FUNCTION_BLOCK CmdCAerationValves (* CAT Function Block Type *)
  (* Standard: 61499-2 *)
  (* Version 0.0, 6/8/2026, Schneider Electric, template *)
  PACKAGE SE.Nereda;
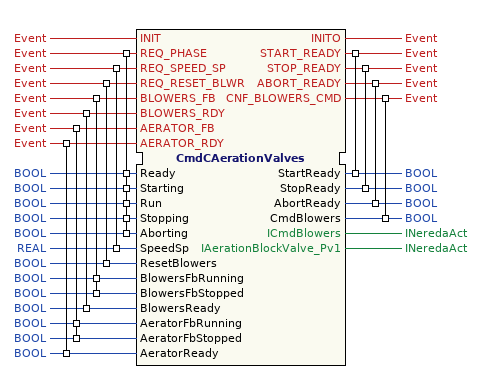
  EVENT_INPUT
    INIT;
    REQ_PHASE WITH Ready, Starting, Run, Stopping, Aborting;
    REQ_SPEED_SP WITH SpeedSp;
    REQ_RESET_BLWR WITH ResetBlowers;
    BLOWERS_FB WITH BlowersFbRunning, BlowersFbStopped;
    BLOWERS_RDY WITH BlowersReady;
    AERATOR_FB WITH AeratorFbRunning, AeratorFbStopped;
    AERATOR_RDY WITH AeratorReady;
  END_EVENT
  EVENT_OUTPUT
    INITO;
    START_READY WITH StartReady;
    STOP_READY WITH StopReady;
    ABORT_READY WITH AbortReady;
    CNF_BLOWERS_CMD WITH CmdBlowers;
  END_EVENT
  VAR_INPUT
    Ready : BOOL;
    Starting : BOOL;
    Run : BOOL;
    Stopping : BOOL;
    Aborting : BOOL;
    SpeedSp : REAL;
    ResetBlowers : BOOL;
    BlowersFbRunning : BOOL;
    BlowersFbStopped : BOOL;
    BlowersReady : BOOL;
    AeratorFbRunning : BOOL;
    AeratorFbStopped : BOOL;
    AeratorReady : BOOL;
  END_VAR
  VAR_OUTPUT
    StartReady : BOOL;
    StopReady : BOOL;
    AbortReady : BOOL;
    CmdBlowers : BOOL;
  END_VAR
  PLUGS
    ICmdBlowers : INeredaAct;
    IAerationBlockValve_Pv1 : INeredaAct;
  END_PLUGS
  (* 01 - FUNCTIONNAL INPUT INTERFACE *)
  (* 00 - INITIALIZATION *)
  (* 05 - LOGIC *)
  (* 06 - HMI INTERFACE *)
  (* 03 - FIELD INTERFACE *)
  (* 02 - FUNCTIONNAL OUTPUT INTERFACE *)
  (* Command Logic *)
  FBS
    IThis : CmdCAerationValves_HMI(QI := TRUE);
    CmdBlowersSmooth : boolValueChanged;
    FbRunBlowers : DS_SELECTX_2536758B411A6CE51; {SET_ATTRIBUTE(Configuration.GenericFBType.InterfaceParams, Runtime.Standard#CNTX:=2;CNTY:=1;DI${CNTX,_,CNTY$}:BOOL)}
    FbStopBlowers : DS_SELECTX_2536758B411A6CE51; {SET_ATTRIBUTE(Configuration.GenericFBType.InterfaceParams, Runtime.Standard#CNTX:=2;CNTY:=1;DI${CNTX,_,CNTY$}:BOOL)}
    FbReadyBlowers : DS_SELECTX_2536758B411A6CE51; {SET_ATTRIBUTE(Configuration.GenericFBType.InterfaceParams, Runtime.Standard#CNTX:=2;CNTY:=1;DI${CNTX,_,CNTY$}:BOOL)}
    BlowersCmd : BOOL2INT;
    CmdLogic : CmdCAerationValvesBasic;
    CmdAerationSmooth : boolValueChanged;
    AerationCmd : BOOL2INT;
    FbRunAerator : DS_SELECTX_2536758B411A6CE51; {SET_ATTRIBUTE(Configuration.GenericFBType.InterfaceParams, Runtime.Standard#CNTX:=2;CNTY:=1;DI${CNTX,_,CNTY$}:BOOL)}
    FbStopAerator : DS_SELECTX_2536758B411A6CE51; {SET_ATTRIBUTE(Configuration.GenericFBType.InterfaceParams, Runtime.Standard#CNTX:=2;CNTY:=1;DI${CNTX,_,CNTY$}:BOOL)}
    FbReadyAerator : DS_SELECTX_2536758B411A6CE51; {SET_ATTRIBUTE(Configuration.GenericFBType.InterfaceParams, Runtime.Standard#CNTX:=2;CNTY:=1;DI${CNTX,_,CNTY$}:BOOL)}
  END_FBS
  EVENT_CONNECTIONS
    INIT TO IThis.3D5D26A512262747;
    IThis.5B84D78EC3FB5466 TO INITO;
    FbRunBlowers.CNF1 TO FbStopBlowers.REQ1;
    FbRunBlowers.CNF2 TO FbStopBlowers.REQ2;
    BLOWERS_RDY TO FbReadyBlowers.REQ2;
    BLOWERS_FB TO FbRunBlowers.REQ2;
    REQ_PHASE TO CmdLogic.0181C35002D51DB9;
    REQ_PHASE TO CmdLogic.7CF49D36E36F42BF;
    REQ_PHASE TO CmdLogic.270A548115E0D83C;
    REQ_PHASE TO CmdLogic.B01B36972B4703C3;
    REQ_PHASE TO CmdLogic.7D39C1849D7CD2AB;
    REQ_SPEED_SP TO ICmdBlowers.1E00729184986247;
    REQ_RESET_BLWR TO ICmdBlowers.37BBC1F841739733;
    FbStopBlowers.IND TO CmdLogic.BLOWERS_STATE;
    FbReadyBlowers.IND TO CmdLogic.BLOWERS_NO_AVAILABLE;
    CmdLogic.CNF_BLOWERS TO CmdBlowersSmooth.REQ;
    CmdLogic.CNF_START_RDY TO START_READY;
    CmdLogic.CNF_STOP_RDY TO STOP_READY;
    CmdLogic.CNF_ABORT_RDY TO ABORT_READY;
    CmdBlowersSmooth.CHD TO BlowersCmd.DD5870AA881150BB;
    BlowersCmd.6FC99A5BD1C38561 TO ICmdBlowers.0F1CDF9A9B4A227A;
    BlowersCmd.6FC99A5BD1C38561 TO CNF_BLOWERS_CMD;
    ICmdBlowers.9CD053F8408797ED TO FbRunBlowers.REQ1;
    ICmdBlowers.CC753684FA882790 TO FbReadyBlowers.REQ1;
    CmdAerationSmooth.CHD TO AerationCmd.DD5870AA881150BB;
    AerationCmd.6FC99A5BD1C38561 TO IAerationBlockValve_Pv1.0F1CDF9A9B4A227A;
    CmdLogic.029C19F2648B74C2 TO CmdAerationSmooth.REQ;
    IAerationBlockValve_Pv1.CC753684FA882790 TO FbReadyAerator.REQ1;
    IAerationBlockValve_Pv1.9CD053F8408797ED TO FbRunAerator.REQ1;
    FbRunAerator.CNF1 TO FbStopAerator.REQ1;
    FbRunAerator.CNF2 TO FbStopAerator.REQ2;
    AERATOR_FB TO FbRunAerator.REQ2;
    AERATOR_RDY TO FbReadyAerator.REQ2;
    FbStopAerator.IND TO CmdLogic.72D3873B05CB4FA1;
    FbReadyAerator.IND TO CmdLogic.6D817C48E98D93B0;
  END_CONNECTIONS
  DATA_CONNECTIONS
    CmdBlowersSmooth.Output TO CmdBlowers;
    BlowersReady TO FbReadyBlowers.DI2_1;
    BlowersFbRunning TO FbRunBlowers.DI2_1;
    BlowersFbStopped TO FbStopBlowers.DI2_1;
    Ready TO CmdLogic.Ready;
    Starting TO CmdLogic.Starting;
    Run TO CmdLogic.Run;
    Stopping TO CmdLogic.Stopping;
    Aborting TO CmdLogic.Aborting;
    SpeedSp TO ICmdBlowers.1BC103921BBFDA0B;
    ResetBlowers TO ICmdBlowers.EA28053F07575F36;
    FbRunBlowers.OUT1 TO CmdLogic.BlowersFbRunning;
    FbStopBlowers.OUT1 TO CmdLogic.BlowersFbStopped;
    FbReadyBlowers.OUT1 TO CmdLogic.BlowersNotAvailable;
    CmdLogic.Blowers TO CmdBlowersSmooth.Input;
    CmdLogic.StartReady TO StartReady;
    CmdLogic.StopReady TO StopReady;
    CmdLogic.AbortReady TO AbortReady;
    CmdBlowersSmooth.Output TO BlowersCmd.4573FC8F228EB71D;
    BlowersCmd.A6DEF5F9C27C1848 TO ICmdBlowers.710D7FC54EE3F35A;
    ICmdBlowers.D83B5BDEFA4D797C TO FbStopBlowers.DI1_1;
    ICmdBlowers.B762734C094A7162 TO FbRunBlowers.DI1_1;
    ICmdBlowers.8A8A07EFCDA1443C TO FbReadyBlowers.DI1_1;
    AerationCmd.A6DEF5F9C27C1848 TO IAerationBlockValve_Pv1.710D7FC54EE3F35A;
    CmdAerationSmooth.Output TO AerationCmd.4573FC8F228EB71D;
    CmdLogic.B0854A3A88322687 TO CmdAerationSmooth.Input;
    IAerationBlockValve_Pv1.B762734C094A7162 TO FbRunAerator.DI1_1;
    IAerationBlockValve_Pv1.D83B5BDEFA4D797C TO FbStopAerator.DI1_1;
    IAerationBlockValve_Pv1.8A8A07EFCDA1443C TO FbReadyAerator.DI1_1;
    AeratorFbRunning TO FbRunAerator.DI2_1;
    AeratorFbStopped TO FbStopAerator.DI2_1;
    AeratorReady TO FbReadyAerator.DI2_1;
    FbRunAerator.OUT1 TO CmdLogic.21FDD93DD473BFE1;
    FbStopAerator.OUT1 TO CmdLogic.087CCAB553E80A7C;
    FbReadyAerator.OUT1 TO CmdLogic.AB5DEAD009B0E55A;
  END_CONNECTIONS
END_FUNCTION_BLOCK
